Omron CX-Programmer project NewProject (CX-Programmer 9.75)

# PLC NewPLC1: CP1E E20

## Program NewProgram1 (cyclic task 0)

### Section Section1

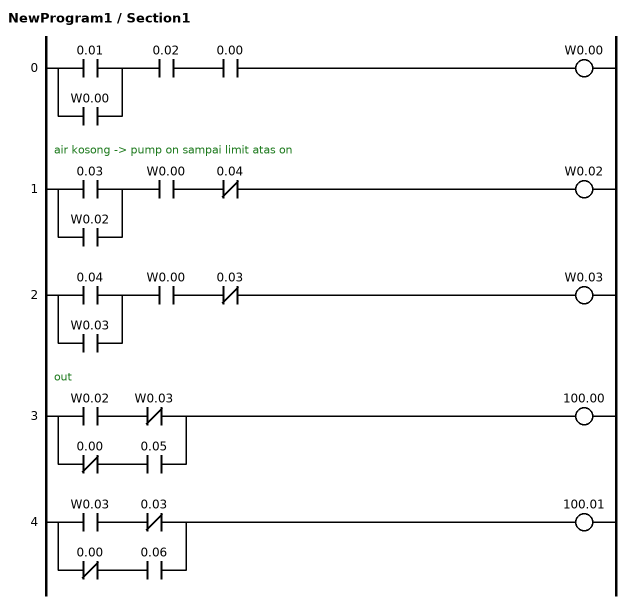
; rung 0
LD 0.01
OR W0.00
AND 0.02
AND 0.00
OUT W0.00
; rung 1: air kosong -> pump on sampai limit atas on
LD 0.03
OR W0.02
AND W0.00
ANDNOT 0.04
OUT W0.02
; rung 2
LD 0.04
OR W0.03
AND W0.00
ANDNOT 0.03
OUT W0.03
; rung 3: out
LD W0.02
ANDNOT W0.03
LDNOT 0.00
AND 0.05
ORLD
OUT 100.00
; rung 4
LD W0.03
ANDNOT 0.03
LDNOT 0.00
AND 0.06
ORLD
OUT 100.01

### Section END
; rung 0
END(001)